PROGRAM Hardware_3300
VAR
    // Servos *********************************************************************
	fbX_Achse										: FB_Achse_NC_PTP_Beckhoff_V2; 
	fbY_Achse										: FB_Achse_NC_PTP_Beckhoff_V2; 

	fbNCI_Channel									: FB_Nc_Kanal;
	
	fbColl_X										: FB_Kollision_1_Achsen;
	fbColl_Y										: FB_Kollision_1_Achsen;

    // Frequenzumrichter **********************************************************
	fbBohraggr_Schluessel_un						: FB_SEW_MOVITRAC_C_CoE;

    // Sensorik *******************************************************************
    fbStillBohraggr_Schluessel_un          			: FB_Belegt;

    // Ventile ********************************************************************
    fbSchluessel_un_Bohrhub                			: FB_Ventil_V2;

    // ***** Hilfsmerker***********************************************************
    (*
        Ventile sind über den DUT_Ventil_para vorparametriert
                ueberwachung_vor_aktiv    : BOOL := TRUE;   // 0 = Endlagenüberwachung vor deaktiviert
                ueberwachung_zur_aktiv    : BOOL := TRUE;   // 0 = Endlagenüberwachung zurück deaktiviert
                ausgang_vor_halten        : BOOL := FALSE;  // 1 = Ausgang immer Ein, sonst 0 in Endlage/1 nicht in Endlage
                ausgang_zur_halten        : BOOL := FALSE;  // 1 = Ausgang immer Ein, sonst 0 in Endlage/1 nicht in Endlage
                entprellen_vor_aktiv      : BOOL := TRUE;   // 0 = Endlage sofort überwachen wenn einmal erreicht
                entprellen_zur_aktiv      : BOOL := TRUE;   // 0 = Endlage sofort überwachen wenn einmal erreicht
                ueberwachungszeit_vor     : TIME := T#10S;  // Überwachungszeit in ms (0-30000ms)
                ueberwachungszeit_zur     : TIME := T#10S;  // Überwachungszeit in ms (0-30000ms)
                entprellungszeit_vor      : TIME := T#50MS; // Entprellungszeit in ms (0-10000ms)
                entprellungszeit_zur      : TIME := T#50MS; // Entprellungszeit in ms (0-10000ms)

        falls etwas anderes gewünscht ist, kann man gezielt für das Ventil die Parameter anpassen
        Beispiel:   ***.para.ausgang_vor_halten := TRUE;
                    ***.para.entprellungszeit_vor := T#100MS;
    *)
END_VAR


// Aktionen aufrufen
//_________________________________________________
	A_Sensorik();
	A_Umrichter();
	A_Ventile();
	A_Servo();
	A_NCI();

ACTION A_NCI:
					
// ***** NCI Kanal *****************************************************************
// *********************************************************************************
	
	GVL_3300.NCI_Steuern.Pfad 		:= 'GVL_0000.Pfad_NCI';
	GVL_3300.NCI_Steuern.PrgName	:= GVL_Visu_3300.aktJob.Programm;
	GVL_3300.NCI_Steuern.Override	:= GVL_Visu_3300.aktJob.Vorschub;
	
	fbNCI_Channel(
		in_Pfad:= GVL_3300.NCI_Steuern.Pfad, 
		in_PName:= GVL_3300.NCI_Steuern.PrgName, 
		in_Override:= GVL_3300.NCI_Steuern.Override, 
		in_NcToPlc:= EAs_3300.e_NCI_Channel, 
		in_nXAxisId	:= 7,
		in_nYAxisId	:= 8,
		in_nZAxisId	:= 0,
		out_PlcToNc=> EAs_3300.a_NCI_Channel, 
		inout_NcReset:= GVL_3300.NCI_Steuern.Reset, 
		inout_PrgLaden:= GVL_3300.NCI_Steuern.PrgLaden, 
		inout_NcGruppe_koppeln:= GVL_3300.NCI_Steuern.Koppeln, 
		inout_NcStart:= GVL_3300.NCI_Steuern.Start, 
		inout_NcStopOverrideNull:= GVL_3300.NCI_Steuern.StopOverrideNull, 
		inout_NcEinzelsatzStart:= GVL_3300.NCI_Steuern.EinzelsatzStart, 
		inout_NcEinzelsatzWeiter:= GVL_3300.NCI_Steuern.EinzelsatzWeiter, 
		inout_NcStatus:= GVL_3300.NCI_Status);
		
		
	GVL_Meldungen.Diagnose_3000.Nr_102	:= UDINT_TO_DINT(fbNCI_Channel.out_FBErrId);	
	GVL_Meldungen.Meldungen_3000.Nr_102 := fbNCI_Channel.out_FBErr ;	
	
	IF fbNCI_Channel.out_FBErr AND GVL_3000.stoerung_quitt THEN
		GVL_3300.NCI_Steuern.Reset := TRUE;
	END_IF
END_ACTION

ACTION A_Sensorik:
					
// ***** Sensorik entprellen *********************************************************
	//********************************************************************************
fbStillBohraggr_Schluessel_un	(	in_Sensor:=,
									in_zeit_aus:=T#100MS,
									in_zeit_aus:=T#100MS,
									Q=>);
END_ACTION

ACTION A_Servo:
					
// ***** Servoregler *****************************************************************
	//********************************************************************************
	GVL_3300.X_Achse_steuern.Reglersperre	:= GVL_3000.bAchsen_Reglersperre;
	GVL_3300.X_Achse_steuern.Freigabe 		:= GVL_3000.bAchsen_Freigabe ;
	
	fbX_Achse(
	in_Reglersperre				:= GVL_3300.X_Achse_steuern.Reglersperre, 
	in_Freigabe					:= GVL_3300.X_Achse_steuern.Freigabe,
	in_Reset					:= GVL_Visu_3300.SteuerStatus.reset   
								OR GVL_3000.stoerung_quitt,                      
	in_Hand						:= GVL_Visu_3300.SteuerStatus.hand,              
	in_Auto						:= GVL_Visu_3300.SteuerStatus.auto,                 
	in_Auto_Override			:= GVL_Visu_3000.override,    
	in_Auto_pos					:= , 
	in_max_Velo					:= 100 ,
	in_PosFenster				:= 0.05, 
	in_Ref_pos					:= 0.0, 
	in_HomingOption				:= , 
	in_EndlageRef				:= , 
	in_DirRef					:= , 
	in_PosEa					:= ,                                       
	out_ist_pos					=> GVL_3300.X_Achse_status.ist_pos, 
	out_in_pos					=> GVL_3300.X_Achse_status.in_pos,   
	out_ziel_pos				=> GVL_3300.X_Achse_status.ziel_pos, 
	out_nicht_ref				=> GVL_3300.X_Achse_status.nicht_ref,      
	out_bremse					=> GVL_3300.X_Achse_status.bremse,           
	out_Achs_Status				=> GVL_3300.X_Achse_status.Achs_Status,  
	inout_NC					:= EAs_3300.ea_X_Achse, 
	inout_service				:= GVL_Visu_3300.X_Achse, 
	inout_Ref_start				:= GVL_3300.X_Achse_steuern.Ref_start, 
	inout_Ref_OK				:= GVL_3300.X_Achse_steuern.Ref_ok, 
	inout_Auto_start			:= GVL_3300.X_Achse_steuern.Auto_start, 
	inout_Auto_stop				:= GVL_3300.X_Achse_steuern.Auto_stop);
	
	GVL_Meldungen.Diagnose_3000.Nr_028	:= fbX_Achse.out_Achs_ErrorID;	
	GVL_Meldungen.Meldungen_3000.Nr_028 := fbX_Achse.out_Achs_Error OR fbX_Achse.out_FB_Error OR fbX_Achse.out_Achs_ErrorID <> 0;		
	GVL_Meldungen.Meldungen_3000.Nr_029 := FALSE;
	GVL_Meldungen.Meldungen_3000.Nr_030 := FALSE;
	//********************************************************************************
					
					
	GVL_3300.Y_Achse_steuern.Reglersperre	:= GVL_3000.bAchsen_Reglersperre;
	GVL_3300.Y_Achse_steuern.Freigabe 		:= GVL_3000.bAchsen_Freigabe;
	
	fbY_Achse(
	in_Reglersperre				:= GVL_3300.Y_Achse_steuern.Reglersperre, 
	in_Freigabe					:= GVL_3300.Y_Achse_steuern.Freigabe,
	in_Reset					:= GVL_Visu_3300.SteuerStatus.reset   
								OR GVL_3000.stoerung_quitt,                      
	in_Hand						:= GVL_Visu_3300.SteuerStatus.hand,              
	in_Auto						:= GVL_Visu_3300.SteuerStatus.auto,                 
	in_Auto_Override			:= GVL_Visu_3000.override,    
	in_Auto_pos					:= , 
	in_max_Velo					:= 100 ,
	in_PosFenster				:= 0.05, 
	in_Ref_pos					:= 0.0, 
	in_HomingOption				:= , 
	in_EndlageRef				:= , 
	in_DirRef					:= , 
	in_PosEa					:= ,                                       
	out_ist_pos					=> GVL_3300.Y_Achse_status.ist_pos, 
	out_in_pos					=> GVL_3300.Y_Achse_status.in_pos,   
	out_ziel_pos				=> GVL_3300.Y_Achse_status.ziel_pos, 
	out_nicht_ref				=> GVL_3300.Y_Achse_status.nicht_ref,      
	out_bremse					=> GVL_3300.Y_Achse_status.bremse,           
	out_Achs_Status				=> GVL_3300.Y_Achse_status.Achs_Status,  
	inout_NC					:= EAs_3300.ea_Y_Achse, 
	inout_service				:= GVL_Visu_3300.Y_Achse, 
	inout_Ref_start				:= GVL_3300.Y_Achse_steuern.Ref_start, 
	inout_Ref_OK				:= GVL_3300.Y_Achse_steuern.Ref_ok, 
	inout_Auto_start			:= GVL_3300.Y_Achse_steuern.Auto_start, 
	inout_Auto_stop				:= GVL_3300.Y_Achse_steuern.Auto_stop);
	
	GVL_Meldungen.Diagnose_3000.Nr_031	:= fbY_Achse.out_Achs_ErrorID;	
	GVL_Meldungen.Meldungen_3000.Nr_031 := fbY_Achse.out_Achs_Error OR fbY_Achse.out_FB_Error OR fbY_Achse.out_Achs_ErrorID <> 0;		
	GVL_Meldungen.Meldungen_3000.Nr_032 := FALSE;
	GVL_Meldungen.Meldungen_3000.Nr_033 := FALSE;

		
	fbColl_X(
		in_Enable := GVL_3000.bAchsen_Freigabe,
		in_Active_Axis_1:= , 
		in_Quittieren:= , 
		in_max_1:= 2790, 
		in_min_1:= -10, 
		in_max_enb:= 90, 
		in_min_enb:= -80, 
		inout_Axis_1:= EAs_3300.ea_X_Achse, 
		out_bError=> );
	
	fbColl_Y(
		in_Enable := GVL_3000.bAchsen_Freigabe,
		in_Active_Axis_1:= , 
		in_Quittieren:= , 
		in_max_1:= 265, 
		in_min_1:= -2, 
		in_max_enb:= 90, 
		in_min_enb:= -80, 
		inout_Axis_1:= EAs_3300.ea_Y_Achse, 
		out_bError=> );
END_ACTION

ACTION A_Umrichter:
	
// ***** Frequenzumrichter ******************************************************
// ******************************************************************************
	GVL_Visu_3300.Bohraggr_Schluessel_un	.Para.Einheit			:= 1;
	GVL_Visu_3300.Bohraggr_Schluessel_un	.Para.Kommastelle		:= 0;

	fbBohraggr_Schluessel_un	(	PD_IN	:=EAs_3300.e_Bohraggr_Schluessel_un	,
			IN_ReglerSperre			:=NOT GVL_3000.bAchsen_Reglersperre,
			IN_SteuerStatus			:=GVL_Visu_3300.SteuerStatus,
			IN_Ethercat_Adresse		:=,
			IN_Ethercat_Name		:='',
			IN_QUITTIEREN			:= GVL_3000.stoerung_quitt,
			IN_OVERRIDE				:= GVL_Visu_3000.override,
			PD_OUT					=> EAs_3300.a_Bohraggr_Schluessel_un	,
			OUT_Stoerung			=> GVL_Meldungen.Meldungen_3000.Nr_006,
			OUT_Fehlernummer		=> GVL_Meldungen.Diagnose_3000.Nr_006,
			OUT_Status				=> GVL_3300.Bohraggr_Schluessel_un_status,
			inout_visu				:= GVL_Visu_3300.Bohraggr_Schluessel_un	,
			inout_steuern			:= GVL_3300.Bohraggr_Schluessel_un_steuern);
	
			GVL_3300.Bohraggr_Schluessel_un_steuern.vor := FALSE;
			GVL_3300.Bohraggr_Schluessel_un_steuern.zur := FALSE;
			GVL_3300.Bohraggr_Schluessel_un_steuern.speed := GVL_Visu_3000.para_Fraeser_Speed_Auto;
END_ACTION

ACTION A_Ventile:
	
// ***** Ventile *********************************************************************
	//********************************************************************************	
	
	GVL_3300.Schluessel_un_Bohrhub.in_freigabe_vor := GVL_3000.bDruckluft_Bereit;
	GVL_3300.Schluessel_un_Bohrhub.in_freigabe_zur := GVL_3000.bDruckluft_Bereit;
	GVL_Visu_3300.Schluessel_un_Bohrhub.para.ausgang_vor_halten:=TRUE;	
	GVL_Visu_3300.Schluessel_un_Bohrhub.para.ausgang_zur_halten:=TRUE;	
	GVL_Visu_3300.Schluessel_un_Bohrhub.para.ueberwachung_vor_aktiv:=TRUE;	
	GVL_Visu_3300.Schluessel_un_Bohrhub.para.ueberwachung_zur_aktiv:=TRUE;	
	GVL_Visu_3300.Schluessel_un_Bohrhub.para.entprellungszeit_vor:=T#50mS;	
	GVL_Visu_3300.Schluessel_un_Bohrhub.para.entprellungszeit_zur:=T#50MS;	
	fbSchluessel_un_Bohrhub (	in_endlage_vor:= EAs_3300.e_FR_3300_Druecker_Schluesselloch_unten_Bohraggregat_6_Bohrhub_ist_oben,
								in_endlage_zur:= EAs_3300.e_FR_3300_Druecker_Schluesselloch_unten_Bohraggregat_6_Bohrhub_ist_unten,
								in_hand:=GVL_Visu_3300.SteuerStatus.hand,
								in_auto:=GVL_Visu_3300.SteuerStatus.auto,
								in_simu :=GVL_3000.bMode_Sim_Ventile,
								in_quit:=GVL_Visu_3300.SteuerStatus.reset 
								OR GVL_3000.stoerung_quitt,
								out_vor=>EAs_3300.a_FR_3300_Druecker_Schluesselloch_unten_Bohraggregat_6_Bohrhub_heben,
								out_zur=>EAs_3300.a_FR_3300_Druecker_Schluesselloch_unten_Bohraggregat_6_Bohrhub_senken,
								out_stoerung_vor=> GVL_Meldungen.Meldungen_3000.Nr_067,
								out_stoerung_zur=> GVL_Meldungen.Meldungen_3000.Nr_068,
								out_stoerung_vorzur=> GVL_Meldungen.Meldungen_3000.Nr_069,
								inout_ansteuerung:=GVL_3300.Schluessel_un_Bohrhub ,
								inout_visu:=GVL_Visu_3300.Schluessel_un_Bohrhub );
END_ACTION

END_PROGRAM

(* stored: Version 1.1.0.1
   POU Hardware_3300: Id {c6e01b9e-323a-4d04-a15e-e3f8d0a1eb00}, SpecialFunc None
   Action A_NCI: Id {c14897c2-9f63-498d-8ff9-d9c16b3e8cc5}
   Action A_Sensorik: Id {4b0b13a8-1aae-4af9-8bd6-839f84eb8833}
   Action A_Servo: Id {123b42bd-40cd-489b-aa99-c7876b679040}
   Action A_Umrichter: Id {76dc17e2-a269-4655-bcc1-2e0c4a948b33}
   Action A_Ventile: Id {4489784c-ae24-4d48-927b-f3db99c24c52} *)
